% RSLogix 500 project MultipositionServoApplication.RSS, saved by version 8.30.00.16 %
PROJECT "UNTITLED"    % processor: Bul.1763 MicroLogix 1100 Series B %

PROGRAM FILES
  LAD 2 "MAIN"  4 rungs
  LAD 3 "IO"  7 rungs
  LAD 4 "CTRL"  11 rungs
  LAD 5 "POSITION"  10 rungs

DATA FILES
  O0 OUTPUT  4 elements
  I1 INPUT  6 elements
  S2 STATUS  66 elements
  B3 BINARY  1 elements
  T4 TIMER  1 elements
  C5 COUNTER  1 elements
  R6 CONTROL  1 elements
  N7 INTEGER  1 elements
  F8 FLOAT  1 elements

LADDER 2 "MAIN"
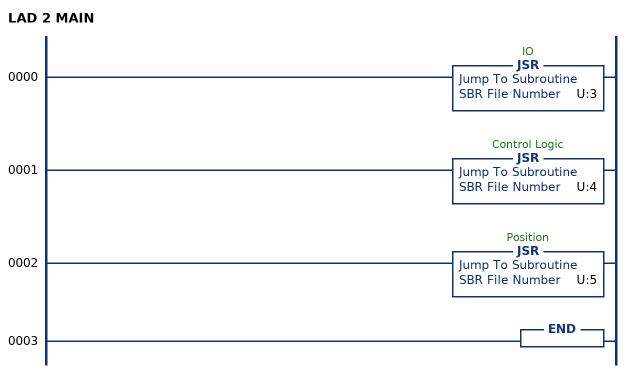
% Rung: 0 %  % edit flag set %
SOR JSR U:3 EOR
%   U:3  "IO" %
% Rung: 1 %  % edit flag set %
SOR JSR U:4 EOR
%   U:4  "Control Logic" %
% Rung: 2 %  % edit flag set %
SOR JSR U:5 EOR
%   U:5  "Position" %
% Rung: 3 %
SOR END EOR

LADDER 3 "IO"
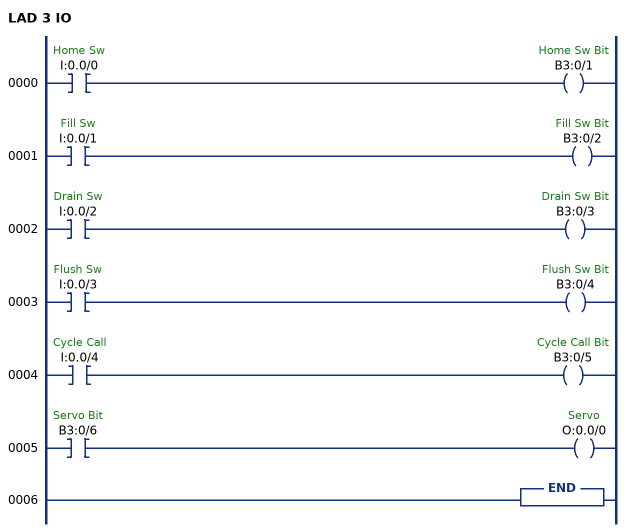
% Rung: 0 %  % edit flag set %
SOR XIC I:0.0/0 OTE B3:0/1 EOR
%   I:0.0/0  "Home Sw" %
%   B3:0/1  "Home Sw Bit" %
% Rung: 1 %  % edit flag set %
SOR XIC I:0.0/1 OTE B3:0/2 EOR
%   I:0.0/1  "Fill Sw" %
%   B3:0/2  "Fill Sw Bit" %
% Rung: 2 %  % edit flag set %
SOR XIC I:0.0/2 OTE B3:0/3 EOR
%   I:0.0/2  "Drain Sw" %
%   B3:0/3  "Drain Sw Bit" %
% Rung: 3 %  % edit flag set %
SOR XIC I:0.0/3 OTE B3:0/4 EOR
%   I:0.0/3  "Flush Sw" %
%   B3:0/4  "Flush Sw Bit" %
% Rung: 4 %  % edit flag set %
SOR XIC I:0.0/4 OTE B3:0/5 EOR
%   I:0.0/4  "Cycle Call" %
%   B3:0/5  "Cycle Call Bit" %
% Rung: 5 %  % edit flag set %
SOR XIC B3:0/6 OTE O:0.0/0 EOR
%   B3:0/6  "Servo Bit" %
%   O:0.0/0  "Servo" %
% Rung: 6 %
SOR END EOR

LADDER 4 "CTRL"
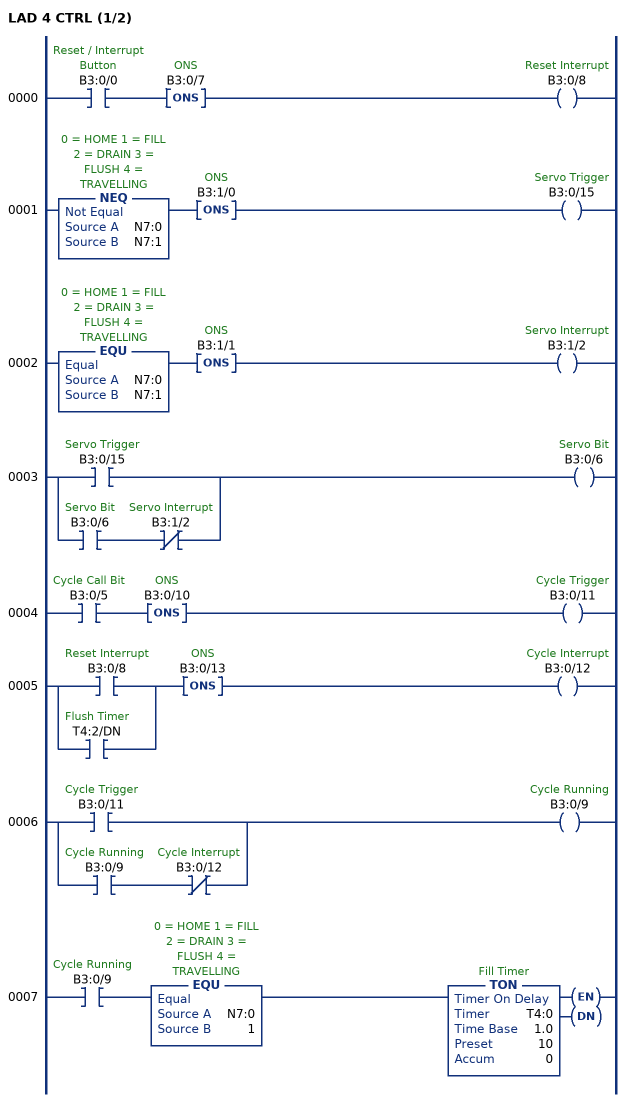
% Rung: 0 %  % edit flag set %
SOR XIC B3:0/0 ONS B3:0/7 OTE B3:0/8 EOR
%   B3:0/0  "Reset / Interrupt Button" %
%   B3:0/7  "ONS" %
%   B3:0/8  "Reset Interrupt" %
% Rung: 1 %  % edit flag set %
SOR NEQ N7:0 N7:1 ONS B3:1/0 OTE B3:0/15 EOR
%   N7:0  "0 = HOME 1 = FILL 2 = DRAIN 3 = FLUSH 4 = TRAVELLING" %
%   N7:1  "Desired: 0 = HOME 1 = FILL 2 = DRAIN 3 = FLUSH" %
%   B3:1/0  "ONS" %
%   B3:0/15  "Servo Trigger" %
% Rung: 2 %  % edit flag set %
SOR EQU N7:0 N7:1 ONS B3:1/1 OTE B3:1/2 EOR
%   N7:0  "0 = HOME 1 = FILL 2 = DRAIN 3 = FLUSH 4 = TRAVELLING" %
%   N7:1  "Desired: 0 = HOME 1 = FILL 2 = DRAIN 3 = FLUSH" %
%   B3:1/1  "ONS" %
%   B3:1/2  "Servo Interrupt" %
% Rung: 3 %  % edit flag set %
SOR BST XIC B3:0/15 NXB XIC B3:0/6 XIO B3:1/2 BND OTE B3:0/6 EOR
%   B3:0/15  "Servo Trigger" %
%   B3:0/6  "Servo Bit" %
%   B3:1/2  "Servo Interrupt" %
% Rung: 4 %  % edit flag set %
SOR XIC B3:0/5 ONS B3:0/10 OTE B3:0/11 EOR
%   B3:0/5  "Cycle Call Bit" %
%   B3:0/10  "ONS" %
%   B3:0/11  "Cycle Trigger" %
% Rung: 5 %  % edit flag set %
SOR BST XIC B3:0/8 NXB XIC T4:2/DN BND ONS B3:0/13 OTE B3:0/12 EOR
%   B3:0/8  "Reset Interrupt" %
%   T4:2  "Flush Timer" %
%   B3:0/13  "ONS" %
%   B3:0/12  "Cycle Interrupt" %
% Rung: 6 %  % edit flag set %
SOR BST XIC B3:0/11 NXB XIC B3:0/9 XIO B3:0/12 BND OTE B3:0/9 EOR
%   B3:0/11  "Cycle Trigger" %
%   B3:0/9  "Cycle Running" %
%   B3:0/12  "Cycle Interrupt" %
% Rung: 7 %  % edit flag set %
SOR XIC B3:0/9 EQU N7:0 1 TON T4:0 1.0 10 0 EOR
%   B3:0/9  "Cycle Running" %
%   N7:0  "0 = HOME 1 = FILL 2 = DRAIN 3 = FLUSH 4 = TRAVELLING" %
%   T4:0  "Fill Timer" %

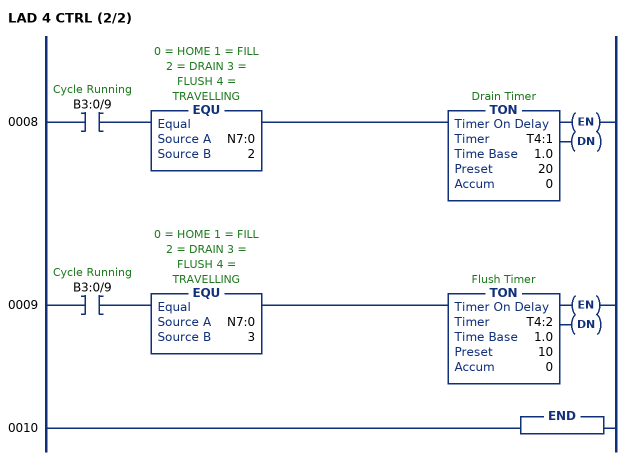
% Rung: 8 %  % edit flag set %
SOR XIC B3:0/9 EQU N7:0 2 TON T4:1 1.0 20 0 EOR
%   B3:0/9  "Cycle Running" %
%   N7:0  "0 = HOME 1 = FILL 2 = DRAIN 3 = FLUSH 4 = TRAVELLING" %
%   T4:1  "Drain Timer" %
% Rung: 9 %  % edit flag set %
SOR XIC B3:0/9 EQU N7:0 3 TON T4:2 1.0 10 0 EOR
%   B3:0/9  "Cycle Running" %
%   N7:0  "0 = HOME 1 = FILL 2 = DRAIN 3 = FLUSH 4 = TRAVELLING" %
%   T4:2  "Flush Timer" %
% Rung: 10 %
SOR END EOR

LADDER 5 "POSITION"
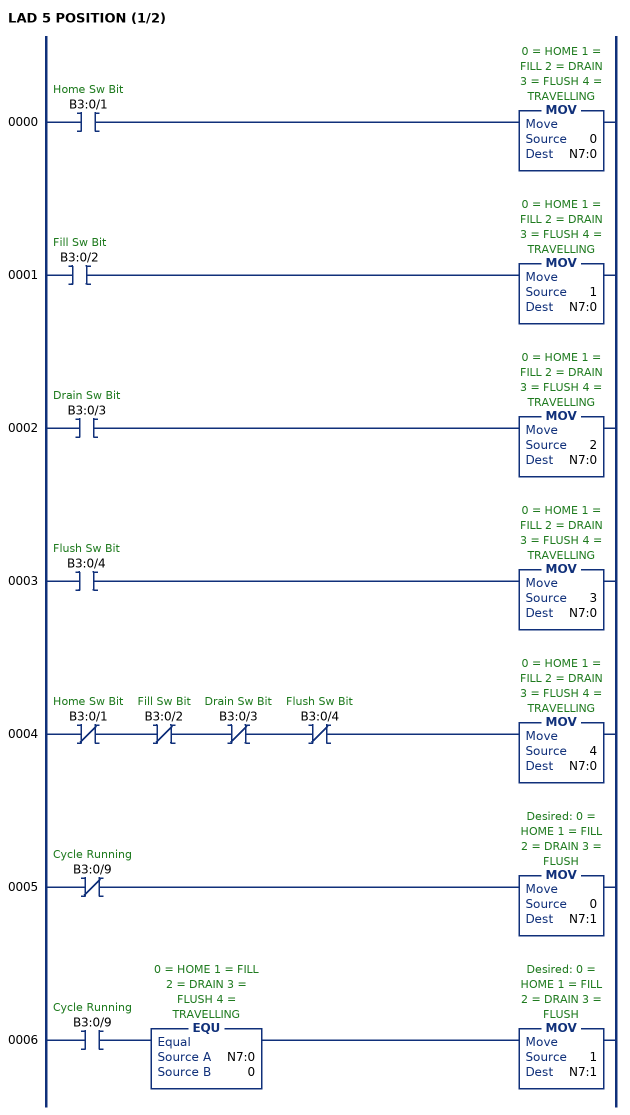
% Rung: 0 %  % edit flag set %
SOR XIC B3:0/1 MOV 0 N7:0 EOR
%   B3:0/1  "Home Sw Bit" %
%   N7:0  "0 = HOME 1 = FILL 2 = DRAIN 3 = FLUSH 4 = TRAVELLING" %
% Rung: 1 %  % edit flag set %
SOR XIC B3:0/2 MOV 1 N7:0 EOR
%   B3:0/2  "Fill Sw Bit" %
%   N7:0  "0 = HOME 1 = FILL 2 = DRAIN 3 = FLUSH 4 = TRAVELLING" %
% Rung: 2 %  % edit flag set %
SOR XIC B3:0/3 MOV 2 N7:0 EOR
%   B3:0/3  "Drain Sw Bit" %
%   N7:0  "0 = HOME 1 = FILL 2 = DRAIN 3 = FLUSH 4 = TRAVELLING" %
% Rung: 3 %  % edit flag set %
SOR XIC B3:0/4 MOV 3 N7:0 EOR
%   B3:0/4  "Flush Sw Bit" %
%   N7:0  "0 = HOME 1 = FILL 2 = DRAIN 3 = FLUSH 4 = TRAVELLING" %
% Rung: 4 %  % edit flag set %
SOR XIO B3:0/1 XIO B3:0/2 XIO B3:0/3 XIO B3:0/4 MOV 4 N7:0 EOR
%   B3:0/1  "Home Sw Bit" %
%   B3:0/2  "Fill Sw Bit" %
%   B3:0/3  "Drain Sw Bit" %
%   B3:0/4  "Flush Sw Bit" %
%   N7:0  "0 = HOME 1 = FILL 2 = DRAIN 3 = FLUSH 4 = TRAVELLING" %
% Rung: 5 %  % edit flag set %
SOR XIO B3:0/9 MOV 0 N7:1 EOR
%   B3:0/9  "Cycle Running" %
%   N7:1  "Desired: 0 = HOME 1 = FILL 2 = DRAIN 3 = FLUSH" %
% Rung: 6 %  % edit flag set %
SOR XIC B3:0/9 EQU N7:0 0 MOV 1 N7:1 EOR
%   B3:0/9  "Cycle Running" %
%   N7:0  "0 = HOME 1 = FILL 2 = DRAIN 3 = FLUSH 4 = TRAVELLING" %
%   N7:1  "Desired: 0 = HOME 1 = FILL 2 = DRAIN 3 = FLUSH" %

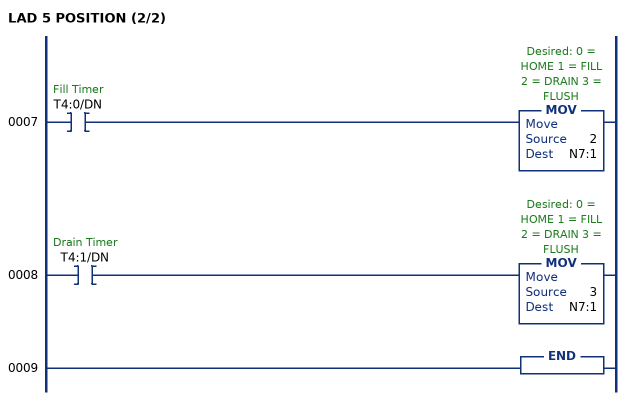
% Rung: 7 %  % edit flag set %
SOR XIC T4:0/DN MOV 2 N7:1 EOR
%   T4:0  "Fill Timer" %
%   N7:1  "Desired: 0 = HOME 1 = FILL 2 = DRAIN 3 = FLUSH" %
% Rung: 8 %  % edit flag set %
SOR XIC T4:1/DN MOV 3 N7:1 EOR
%   T4:1  "Drain Timer" %
%   N7:1  "Desired: 0 = HOME 1 = FILL 2 = DRAIN 3 = FLUSH" %
% Rung: 9 %
SOR END EOR

OTHER DOCUMENTED ADDRESSES
  B3:0/14  "Cycle Complete"
  B3:2/0  "ONS"
